Fanuc KAREL source: kx00003.KL

PROGRAM KX00003
%STACKSIZE=65535
%PRIORITY=65535
%NOLOCKGROUP
VAR
I : INTEGER
J : INTEGER
B : BOOLEAN
F : FILE
S : STRING[80]
P : XYZWPR
BEGIN
OPEN FILE F ('RW','MD:KFSAMPLE.DT')
-- UNRESOLVED_PC line 12 opcodes [22 3F 9C 9C 37 9C 9C 37 2C] marker_code=32
CLOSE FILE F
END KX00003
